FUNCTION_BLOCK FB_Bel_RGBW_Sued
VAR_INPUT
	Freigabe_auto			: BOOL;
	Freigabe_Deakt_auto		: BOOL;
	Betrieb_Anford_auto		: BOOL;
	Farbcode			: STRING;
	Adresse_R				: BYTE;
	Adresse_G				: BYTE;
	Adresse_B				: BYTE;
	Adresse_W				: BYTE;
	Quittierung				: BOOL;
	AdressType				: E_DALIV2AddrType;
	Reset					: BOOL;

END_VAR
VAR_OUTPUT
	{attribute 'OPC.UA.DA' := '1'}Steuerung				: ST_Bel_Steuerung;			
	{attribute 'OPC.UA.DA' := '1'}Stellwert				: ST_Bel_Stellwert;			
	{attribute 'OPC.UA.DA' := '1'}Zustand					: ST_Bel_Zustand;		
	{attribute 'OPC.UA.DA' := '1'}Parameter				: ST_Bel_Parameter;			
END_VAR
VAR
	Beleuchtung_R			: FB_Bel_Einzel_farbe;
	Beleuchtung_G			: FB_Bel_Einzel_farbe;
	Beleuchtung_B			: FB_Bel_Einzel_farbe;
	Beleuchtung_W			: FB_Bel_Einzel_farbe;

	Stellwert_R_Regelung	: REAL;
	Stellwert_G_Regelung	: REAL;
	Stellwert_B_Regelung	: REAL;
	Stellwert_W_Regelung	: REAL;

	Zustand_Bel_R			: ST_BEL_Zustand;
	Zustand_Bel_G			: ST_BEL_Zustand;
	Zustand_Bel_B			: ST_BEL_Zustand;
	Zustand_Bel_W			: ST_BEL_Zustand;

	Logik					: FB_Bel_RGBW_Logik;
	Ablaufsteuerung			: FB_Bel_RGBW_Ablaufsteuerung;

	Regelung				: FB_Bel_RGBW_Regelung;
	QuitTrig				: FB_SetResetFallTrigger;
	Anschaltung				: BOOL;

	Time_on: TON;
	Reset1: TON;

	Beleuchtung_SW_R: FB_Bel_Einzel_farbe;
END_VAR

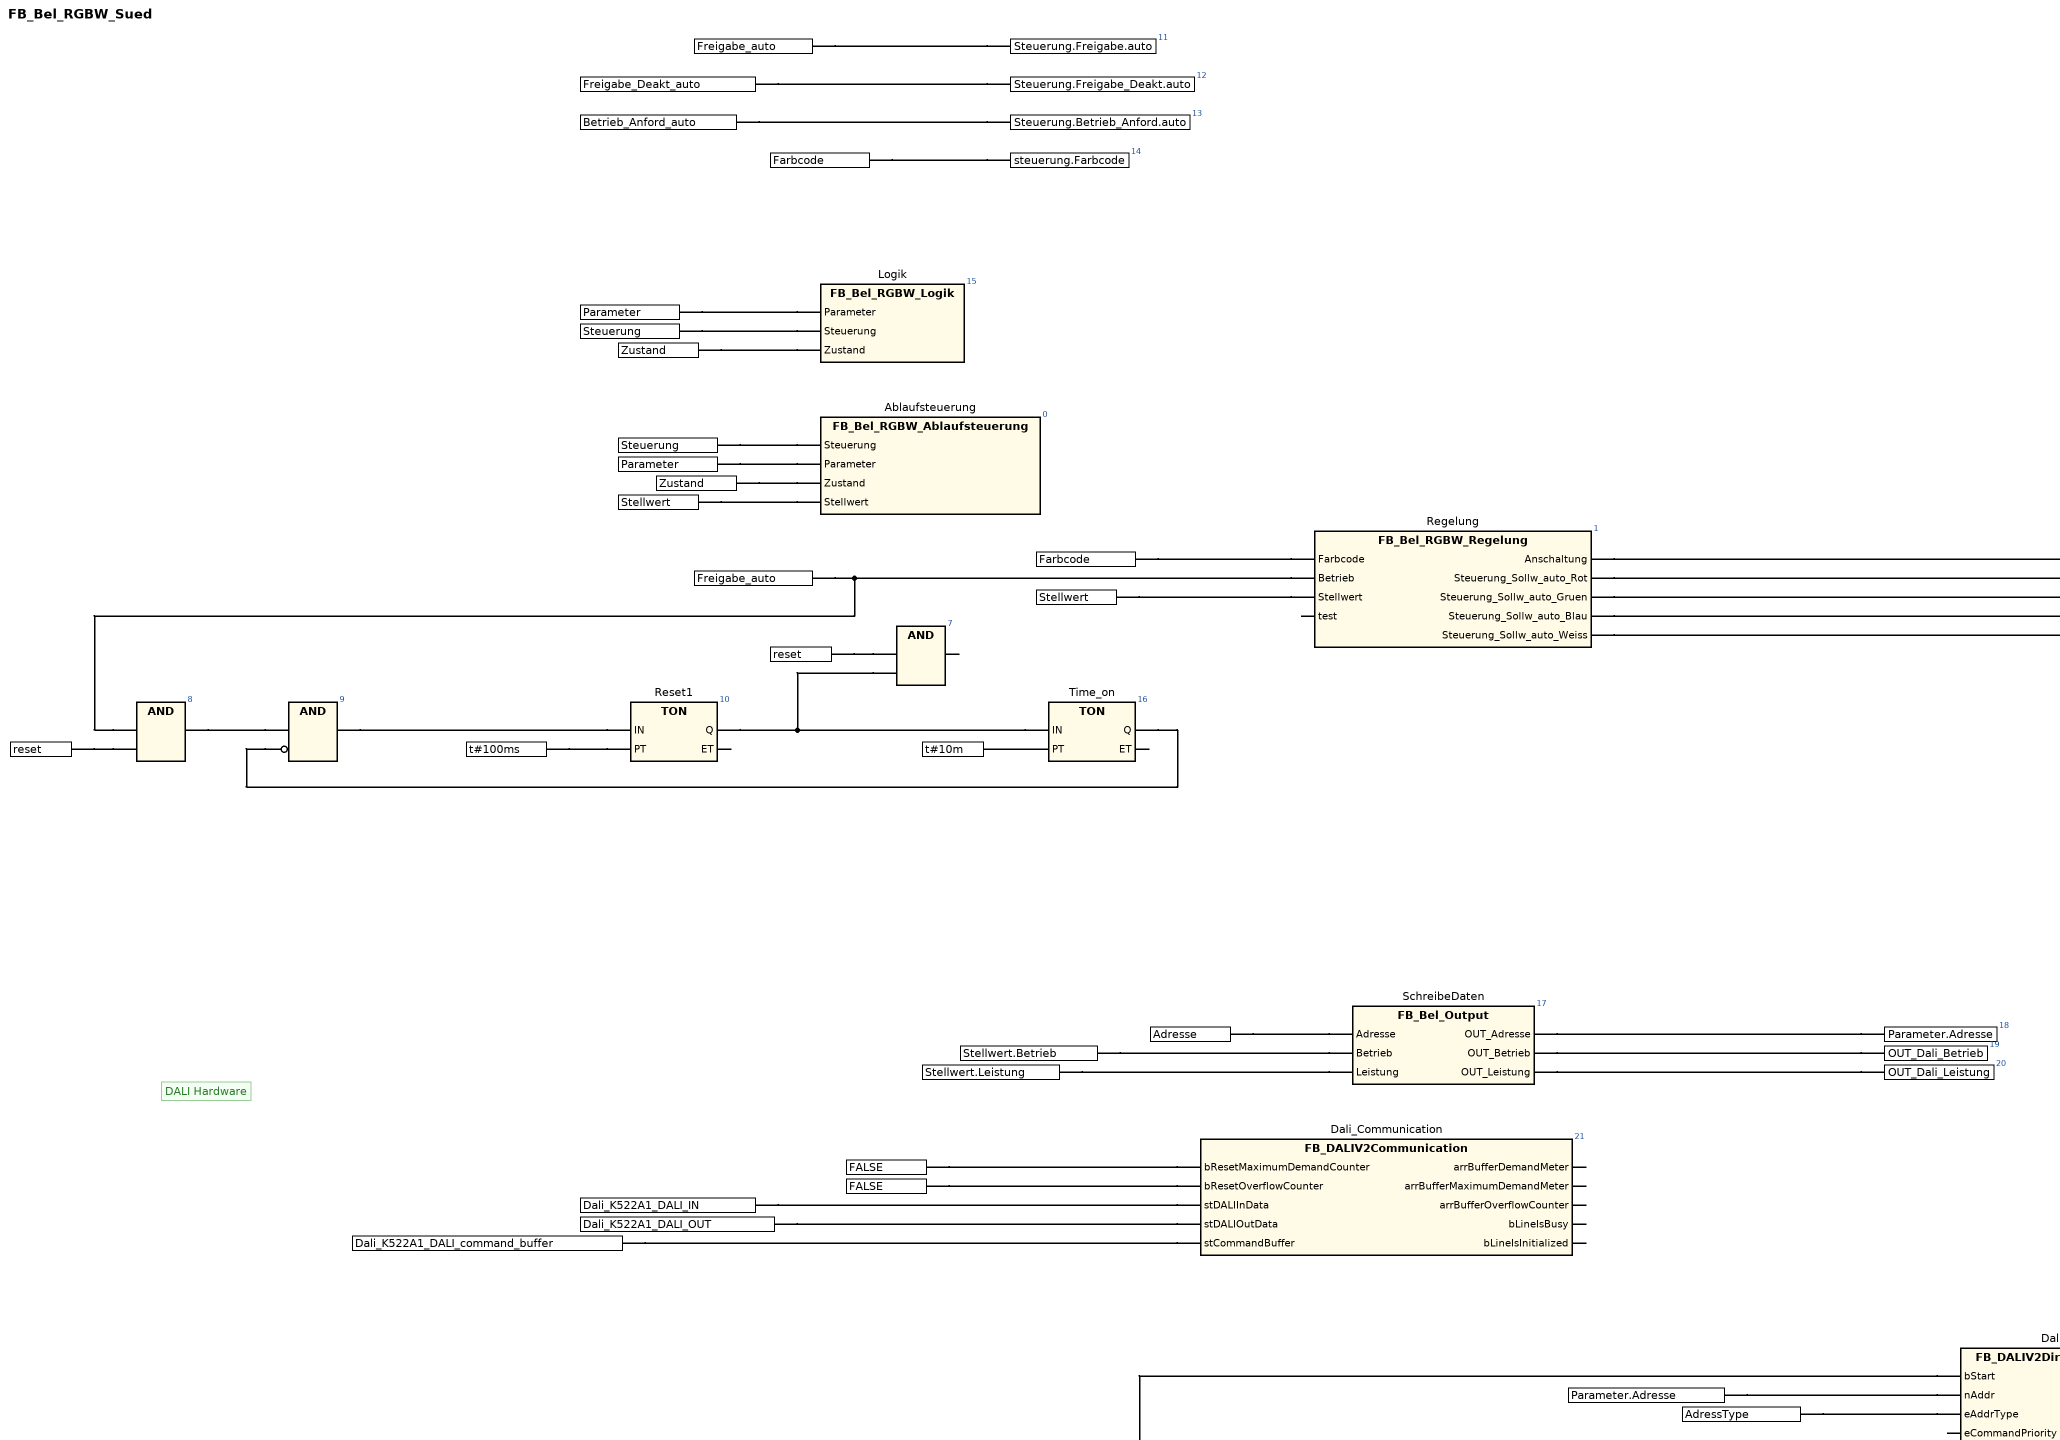
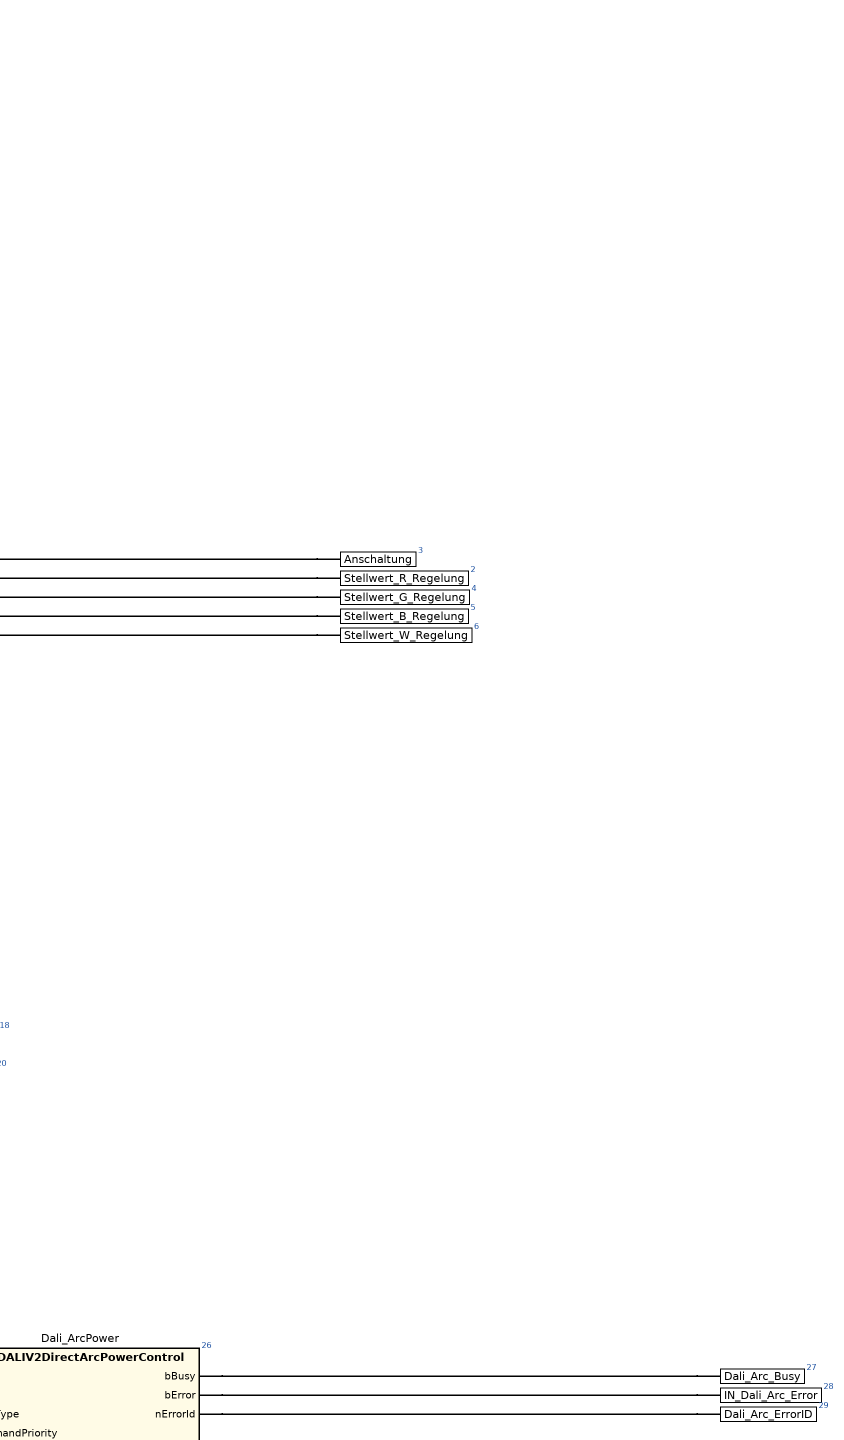
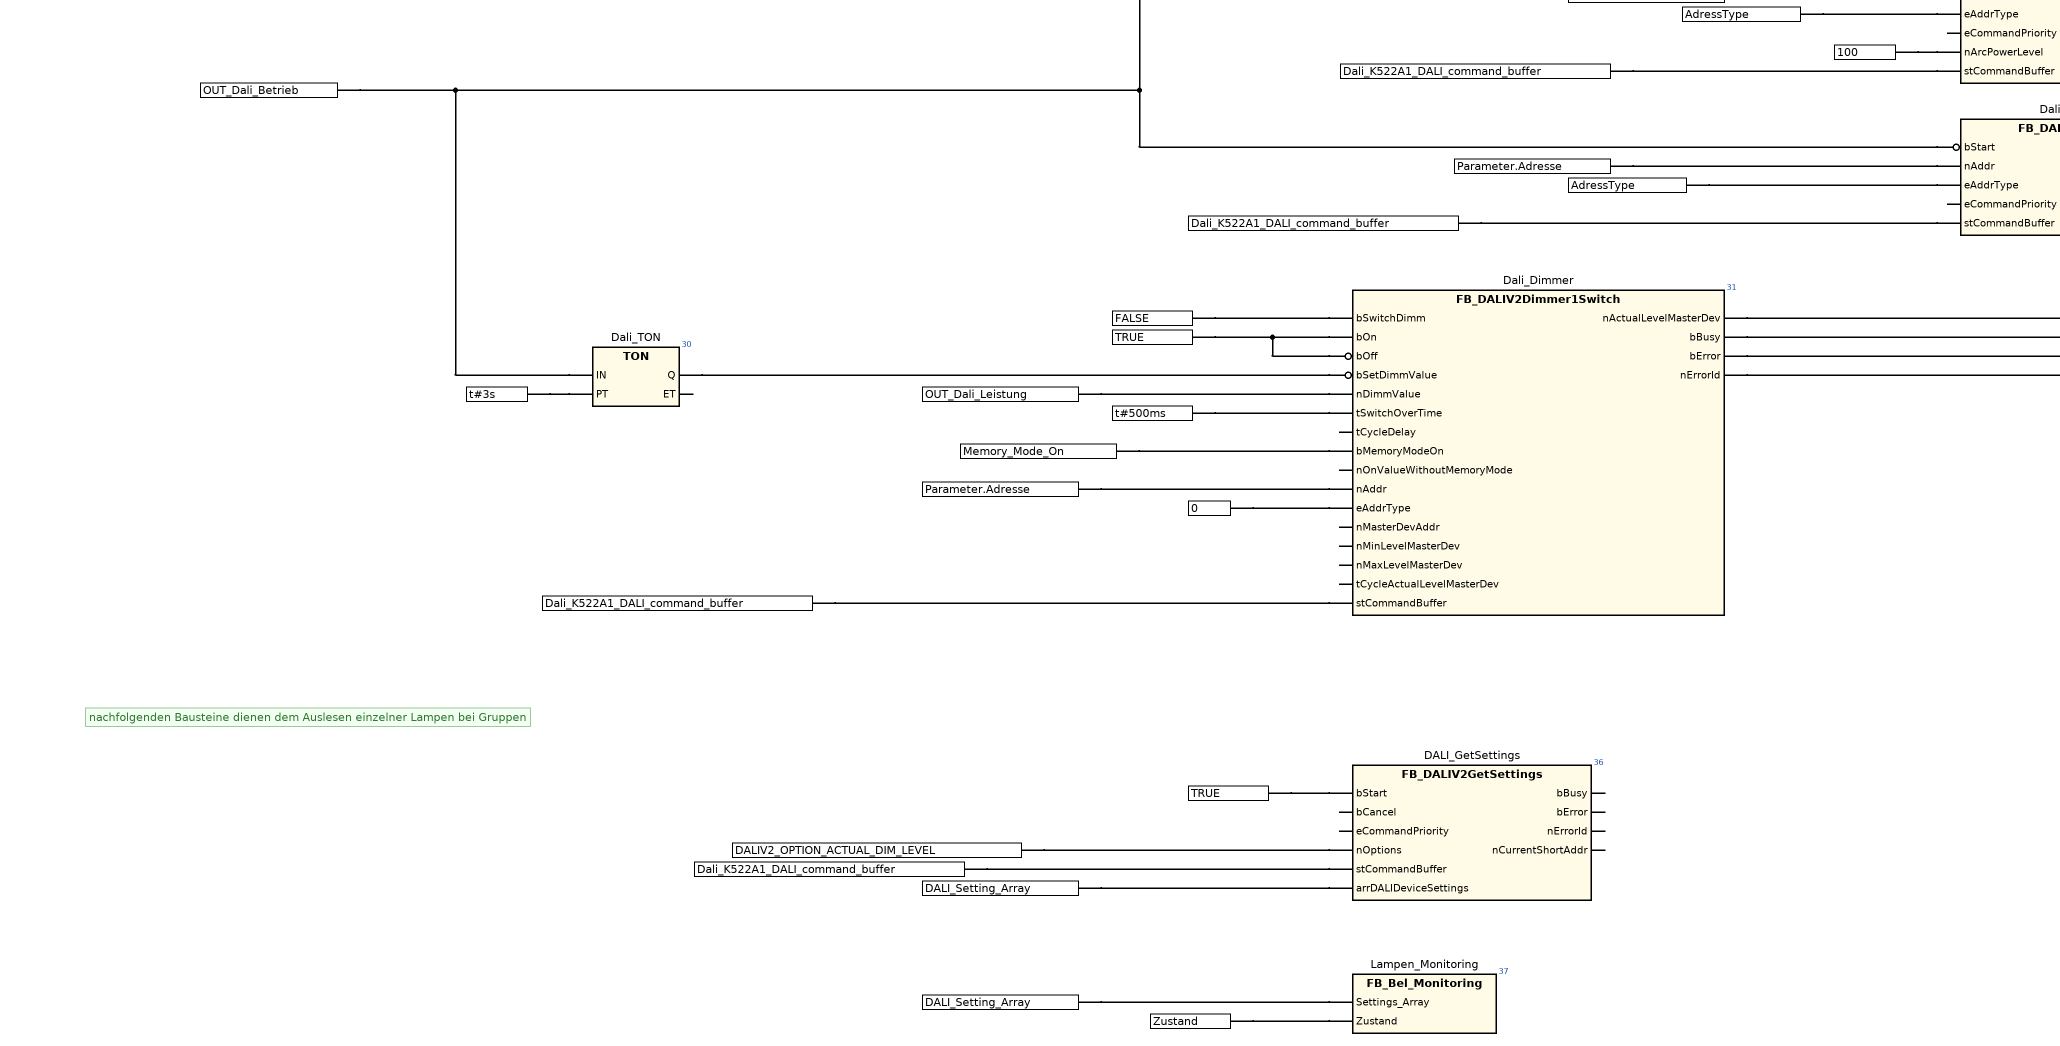
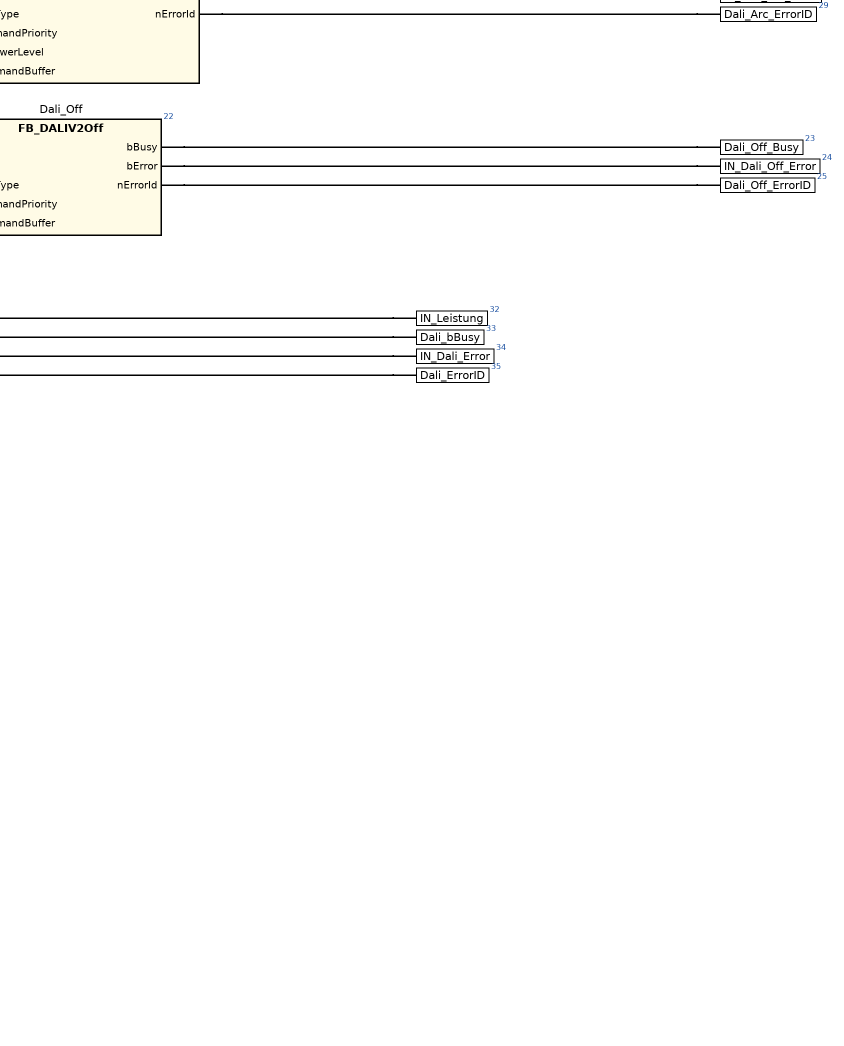
Ablaufsteuerung(Steuerung := Steuerung, Parameter := Parameter, Zustand := Zustand, Stellwert := Stellwert); // FB_Bel_RGBW_Ablaufsteuerung
Regelung(Farbcode := Farbcode, Betrieb := Freigabe_auto, Stellwert := Stellwert); // FB_Bel_RGBW_Regelung
Stellwert_R_Regelung := Regelung.Steuerung_Sollw_auto_Rot;
Anschaltung := Regelung.Anschaltung;
Stellwert_G_Regelung := Regelung.Steuerung_Sollw_auto_Gruen;
Stellwert_B_Regelung := Regelung.Steuerung_Sollw_auto_Blau;
Stellwert_W_Regelung := Regelung.Steuerung_Sollw_auto_Weiss;
(* reset AND Reset1.Q; result not used *)
Reset1(IN := (Freigabe_auto AND reset) AND NOT Time_on.Q, PT := t#100ms); // TON
Steuerung.Freigabe.auto := Freigabe_auto;
Steuerung.Freigabe_Deakt.auto := Freigabe_Deakt_auto;
Steuerung.Betrieb_Anford.auto := Betrieb_Anford_auto;
steuerung.Farbcode := Farbcode;
Logik(Parameter := Parameter, Steuerung := Steuerung, Zustand := Zustand); // FB_Bel_RGBW_Logik
Time_on(IN := Reset1.Q, PT := t#10m); // TON
SchreibeDaten(Adresse := Adresse, Betrieb := Stellwert.Betrieb, Leistung := Stellwert.Leistung); // FB_Bel_Output
Parameter.Adresse := SchreibeDaten.OUT_Adresse;
OUT_Dali_Betrieb := SchreibeDaten.OUT_Betrieb;
OUT_Dali_Leistung := SchreibeDaten.OUT_Leistung;
// DALI Hardware
Dali_Communication(
    bResetMaximumDemandCounter := FALSE,
    bResetOverflowCounter := FALSE,
    stDALIInData := Dali_K522A1_DALI_IN,
    stDALIOutData := Dali_K522A1_DALI_OUT,
    stCommandBuffer := Dali_K522A1_DALI_command_buffer); // FB_DALIV2Communication
Dali_Off(
    bStart := NOT OUT_Dali_Betrieb,
    nAddr := Parameter.Adresse,
    eAddrType := AdressType,
    stCommandBuffer := Dali_K522A1_DALI_command_buffer); // FB_DALIV2Off
Dali_Off_Busy := Dali_Off.bBusy;
IN_Dali_Off_Error := Dali_Off.bError;
Dali_Off_ErrorID := Dali_Off.nErrorId;
Dali_ArcPower(
    bStart := OUT_Dali_Betrieb,
    nAddr := Parameter.Adresse,
    eAddrType := AdressType,
    nArcPowerLevel := 100,
    stCommandBuffer := Dali_K522A1_DALI_command_buffer); // FB_DALIV2DirectArcPowerControl
Dali_Arc_Busy := Dali_ArcPower.bBusy;
IN_Dali_Arc_Error := Dali_ArcPower.bError;
Dali_Arc_ErrorID := Dali_ArcPower.nErrorId;
Dali_TON(IN := OUT_Dali_Betrieb, PT := t#3s); // TON
Dali_Dimmer(
    bSwitchDimm := FALSE,
    bOn := TRUE,
    bOff := NOT TRUE,
    bSetDimmValue := NOT Dali_TON.Q,
    nDimmValue := OUT_Dali_Leistung,
    tSwitchOverTime := t#500ms,
    bMemoryModeOn := Memory_Mode_On,
    nAddr := Parameter.Adresse,
    eAddrType := 0,
    stCommandBuffer := Dali_K522A1_DALI_command_buffer); // FB_DALIV2Dimmer1Switch
IN_Leistung := Dali_Dimmer.nActualLevelMasterDev;
Dali_bBusy := Dali_Dimmer.bBusy;
IN_Dali_Error := Dali_Dimmer.bError;
Dali_ErrorID := Dali_Dimmer.nErrorId;
// nachfolgenden Bausteine dienen dem Auslesen einzelner Lampen bei Gruppen
DALI_GetSettings(
    bStart := TRUE,
    nOptions := DALIV2_OPTION_ACTUAL_DIM_LEVEL,
    stCommandBuffer := Dali_K522A1_DALI_command_buffer,
    arrDALIDeviceSettings := DALI_Setting_Array); // FB_DALIV2GetSettings
Lampen_Monitoring(Settings_Array := DALI_Setting_Array, Zustand := Zustand); // FB_Bel_Monitoring

END_FUNCTION_BLOCK

(* stored: Version 1.1.0.1, ProductVersion 3.1.4024.9
   POU FB_Bel_RGBW_Sued: Id {bd01d782-cf30-4031-972b-92c096d98c83}, SpecialFunc None *)
